% RSLogix 500 project LVD4000_ND_CHICAGO_0020711_Mini.RSS, saved by version 11.00.00.00 %
PROJECT "LVD4000"    % processor: MicroLogix 1400 %

PROGRAM FILES
  LAD 2 "MAIN"  31 rungs  % Main Program Routine %
  LAD 3 "BOT HSC"  2 rungs  % Bottom Conveyor High-Speed Counter Routine %
  LAD 4 "TOP HSC"  2 rungs  % Top Conveyor High-Speed Counter Routine %
  LAD 5 "BOT_TRACK"  3 rungs  % Bottom Conveyor Triggering & Tracking Sequence %
  LAD 6 "TOP_TRACK"  3 rungs  % Top Conveyor Triggering & Tracking Sequence %
  LAD 7 "FOR_HMI"  8 rungs
  LAD 8 "BOT_OPTIC"  6 rungs
  LAD 10 "BOT_TOP"  21 rungs
  LAD 12 "BOT_TRANSF"  3 rungs
  LAD 14 "TOP_OPTIC"  12 rungs
  LAD 16 "TOP_SIDE"  24 rungs
  LAD 18 "TOP_PYRIMI"  5 rungs
  LAD 20 "TOP_TOP"  22 rungs
  LAD 22 "TOP_THREAD"  2 rungs
  LAD 24 "TOP_BLOW"  12 rungs
  LAD 26 "FLOW"  15 rungs
  LAD 28 "FAULTS"  26 rungs
  LAD 30 "SPEED"  8 rungs
  LAD 32 "BOXER"  17 rungs
  LAD 34 "CLEANUP"  20 rungs

DATA FILES
  O0 OUTPUT  6 elements
  I1 INPUT  8 elements
  S2 STATUS  66 elements
  B3 BINARY  11 elements
  T4 TIMER  30 elements
  C5 COUNTER  1 elements
  R6 CONTROL  3 elements
  N7 INTEGER  100 elements
  F8 FLOAT  40 elements
  B9   256 elements
  N10 HMI_COM  100 elements
  B11   256 elements
  B12 BOXER_BITS  3 elements
  N16   1 elements
  B18   11 elements
  T20   1 elements
  R21   4 elements
  B22   35 elements

LADDER 2 "MAIN"    % Main Program Routine %
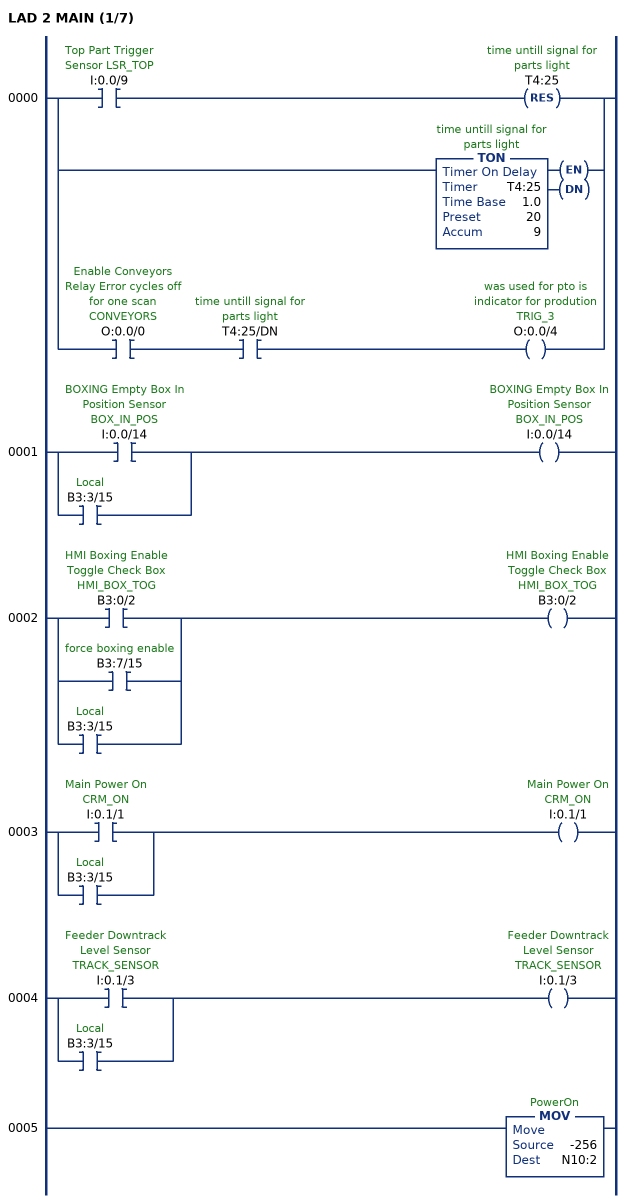
% Rung: 0 %
SOR BST XIC I:0.0/9 RES T4:25 NXB TON T4:25 1.0 20 9 NXB XIC O:0.0/0 XIC T4:25/DN OTE O:0.0/4 BND EOR
%   I:0.0/9  LSR_TOP  "Top Part Trigger Sensor" %
%   T4:25  "time untill signal for parts light" %
%   O:0.0/0  CONVEYORS  "Enable Conveyors Relay Error cycles off for one scan" %
%   O:0.0/4  TRIG_3  "was used for pto is indicator for prodution" %
% Rung: 1 %
SOR BST XIC I:0.0/14 NXB XIC B3:3/15 BND OTE I:0.0/14 EOR
%   I:0.0/14  BOX_IN_POS  "BOXING Empty Box In Position Sensor" %
%   B3:3/15  "Local" %
% Rung: 2 %
SOR BST XIC B3:0/2 NXB XIC B3:7/15 NXB XIC B3:3/15 BND OTE B3:0/2 EOR
%   B3:0/2  HMI_BOX_TOG  "HMI Boxing Enable Toggle Check Box" %
%   B3:7/15  "force boxing enable" %
%   B3:3/15  "Local" %
% Rung: 3 %
SOR BST XIC I:0.1/1 NXB XIC B3:3/15 BND OTE I:0.1/1 EOR
%   I:0.1/1  CRM_ON  "Main Power On" %
%   B3:3/15  "Local" %
% Rung: 4 %
SOR BST XIC I:0.1/3 NXB XIC B3:3/15 BND OTE I:0.1/3 EOR
%   I:0.1/3  TRACK_SENSOR  "Feeder Downtrack Level Sensor" %
%   B3:3/15  "Local" %
% Rung: 5 %
SOR MOV -256 N10:2 EOR
%   N10:2  "PowerOn" %

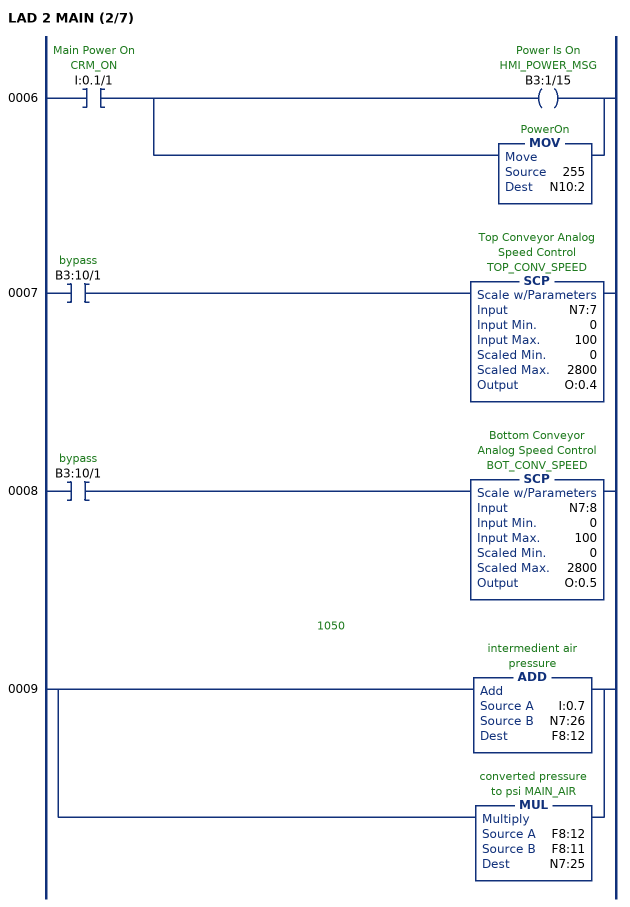
% Rung: 6 %
SOR XIC I:0.1/1 BST OTE B3:1/15 NXB MOV 255 N10:2 BND EOR
%   I:0.1/1  CRM_ON  "Main Power On" %
%   B3:1/15  HMI_POWER_MSG  "Power Is On" %
%   N10:2  "PowerOn" %
% Rung: 7 %
SOR XIC B3:10/1 SCP N7:7 0 100 0 2800 O:0.4 EOR
%   B3:10/1  "bypass" %
%   N7:7  "Top Conv Speed" %
%   O:0.4  TOP_CONV_SPEED  "Top Conveyor Analog Speed Control" %
% Rung: 8 %
SOR XIC B3:10/1 SCP N7:8 0 100 0 2800 O:0.5 EOR
%   B3:10/1  "bypass" %
%   N7:8  "Bottom Conveyor Speed" %
%   O:0.5  BOT_CONV_SPEED  "Bottom Conveyor Analog Speed Control" %
% Rung: 9 %
% 1050 %
SOR BST ADD I:0.7 N7:26 F8:12 NXB MUL F8:12 F8:11 N7:25 BND EOR
%   N7:26  MAIN_AIR_OFFSET  "Main Air Offset" %
%   F8:12  "intermedient air pressure" %
%   F8:11  AIR_MULTIPLIER  "main air multiplyer" %
%   N7:25  MAIN_AIR  "converted pressure to psi" %

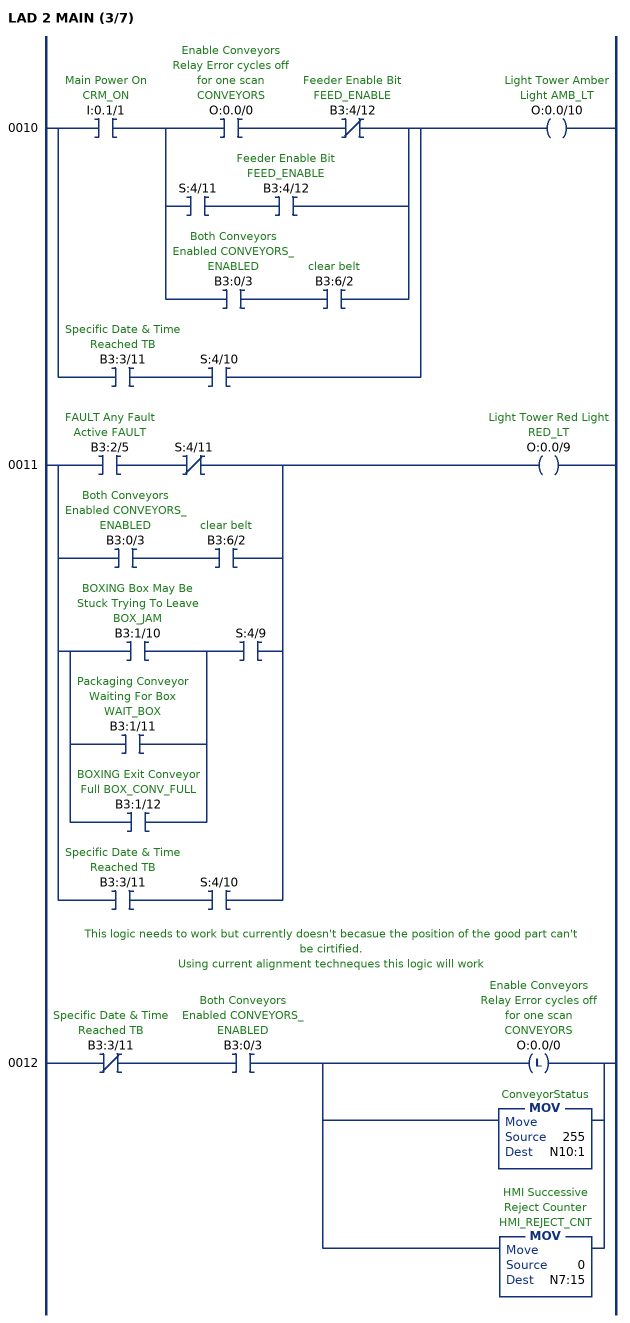
% Rung: 10 %
SOR BST XIC I:0.1/1 BST XIC O:0.0/0 XIO B3:4/12 NXB XIC S:4/11 XIC B3:4/12 NXB XIC B3:0/3 XIC B3:6/2 BND NXB XIC B3:3/11 XIC S:4/10 BND OTE O:0.0/10 EOR
%   I:0.1/1  CRM_ON  "Main Power On" %
%   O:0.0/0  CONVEYORS  "Enable Conveyors Relay Error cycles off for one scan" %
%   B3:4/12  FEED_ENABLE  "Feeder Enable Bit" %
%   B3:0/3  CONVEYORS_ENABLED  "Both Conveyors Enabled" %
%   B3:6/2  "clear belt" %
%   B3:3/11  TB  "Specific Date & Time Reached" %
%   O:0.0/10  AMB_LT  "Light Tower Amber Light" %
% Rung: 11 %
SOR BST BST XIC B3:2/5 XIO S:4/11 NXB XIC B3:0/3 XIC B3:6/2 NXB BST XIC B3:1/10 NXB XIC B3:1/11 NXB XIC B3:1/12 BND XIC S:4/9 BND NXB XIC B3:3/11 XIC S:4/10 BND OTE O:0.0/9 EOR
%   B3:2/5  FAULT  "FAULT Any Fault Active" %
%   B3:0/3  CONVEYORS_ENABLED  "Both Conveyors Enabled" %
%   B3:6/2  "clear belt" %
%   B3:1/10  BOX_JAM  "BOXING Box May Be Stuck Trying To Leave" %
%   B3:1/11  WAIT_BOX  "Packaging Conveyor Waiting For Box" %
%   B3:1/12  BOX_CONV_FULL  "BOXING Exit Conveyor Full" %
%   B3:3/11  TB  "Specific Date & Time Reached" %
%   O:0.0/9  RED_LT  "Light Tower Red Light" %
% Rung: 12 %
% This logic needs to work but currently doesn't becasue the position of the good part can't be cirtified.
% 
% Using current alignment techneques this logic will work %
SOR XIO B3:3/11 XIC B3:0/3 BST OTL O:0.0/0 NXB MOV 255 N10:1 NXB MOV 0 N7:15 BND EOR
%   B3:3/11  TB  "Specific Date & Time Reached" %
%   B3:0/3  CONVEYORS_ENABLED  "Both Conveyors Enabled" %
%   O:0.0/0  CONVEYORS  "Enable Conveyors Relay Error cycles off for one scan" %
%   N10:1  "ConveyorStatus" %
%   N7:15  HMI_REJECT_CNT  "HMI Successive Reject Counter" %

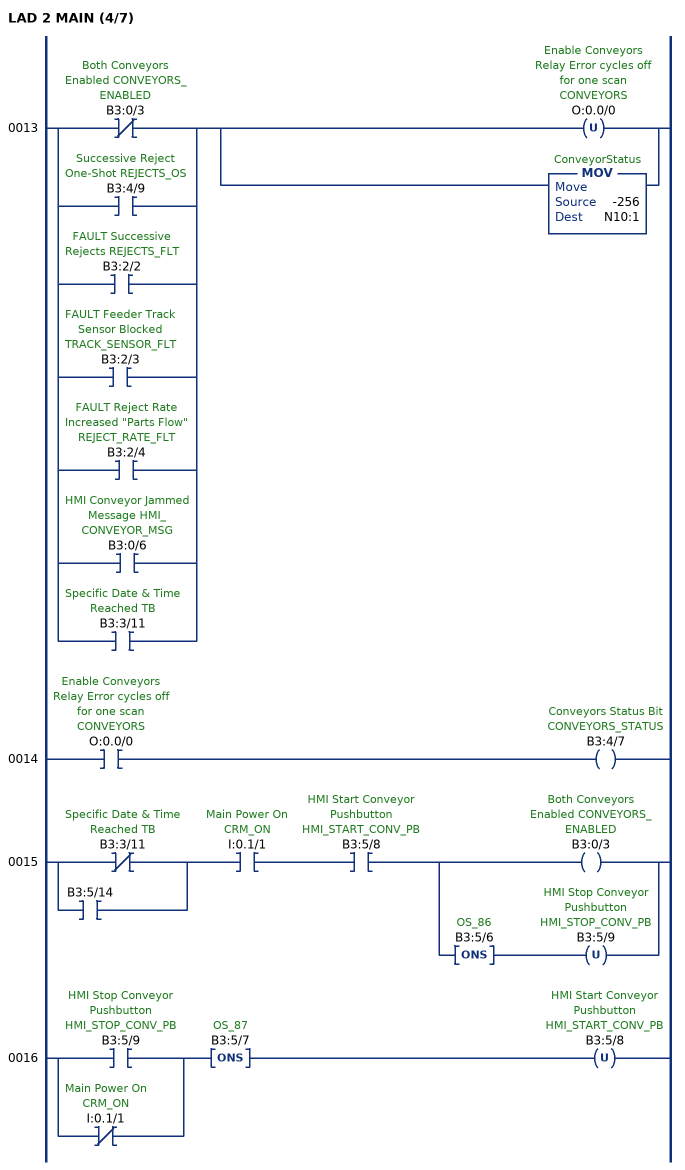
% Rung: 13 %
SOR BST XIO B3:0/3 NXB XIC B3:4/9 NXB XIC B3:2/2 NXB XIC B3:2/3 NXB XIC B3:2/4 NXB XIC B3:0/6 NXB XIC B3:3/11 BND BST OTU O:0.0/0 NXB MOV -256 N10:1 BND EOR
%   B3:0/3  CONVEYORS_ENABLED  "Both Conveyors Enabled" %
%   B3:4/9  REJECTS_OS  "Successive Reject One-Shot" %
%   B3:2/2  REJECTS_FLT  "FAULT Successive Rejects" %
%   B3:2/3  TRACK_SENSOR_FLT  "FAULT Feeder Track Sensor Blocked" %
%   B3:2/4  REJECT_RATE_FLT  "FAULT Reject Rate Increased "Parts Flow"" %
%   B3:0/6  HMI_CONVEYOR_MSG  "HMI Conveyor Jammed Message" %
%   B3:3/11  TB  "Specific Date & Time Reached" %
%   O:0.0/0  CONVEYORS  "Enable Conveyors Relay Error cycles off for one scan" %
%   N10:1  "ConveyorStatus" %
% Rung: 14 %
SOR XIC O:0.0/0 OTE B3:4/7 EOR
%   O:0.0/0  CONVEYORS  "Enable Conveyors Relay Error cycles off for one scan" %
%   B3:4/7  CONVEYORS_STATUS  "Conveyors Status Bit" %
% Rung: 15 %
SOR BST XIO B3:3/11 NXB XIC B3:5/14 BND XIC I:0.1/1 XIC B3:5/8 BST OTE B3:0/3 NXB ONS B3:5/6 OTU B3:5/9 BND EOR
%   B3:3/11  TB  "Specific Date & Time Reached" %
%   I:0.1/1  CRM_ON  "Main Power On" %
%   B3:5/8  HMI_START_CONV_PB  "HMI Start Conveyor Pushbutton" %
%   B3:0/3  CONVEYORS_ENABLED  "Both Conveyors Enabled" %
%   B3:5/6  OS_86 %
%   B3:5/9  HMI_STOP_CONV_PB  "HMI Stop Conveyor Pushbutton" %
% Rung: 16 %
SOR BST XIC B3:5/9 NXB XIO I:0.1/1 BND ONS B3:5/7 OTU B3:5/8 EOR
%   B3:5/9  HMI_STOP_CONV_PB  "HMI Stop Conveyor Pushbutton" %
%   I:0.1/1  CRM_ON  "Main Power On" %
%   B3:5/7  OS_87 %
%   B3:5/8  HMI_START_CONV_PB  "HMI Start Conveyor Pushbutton" %

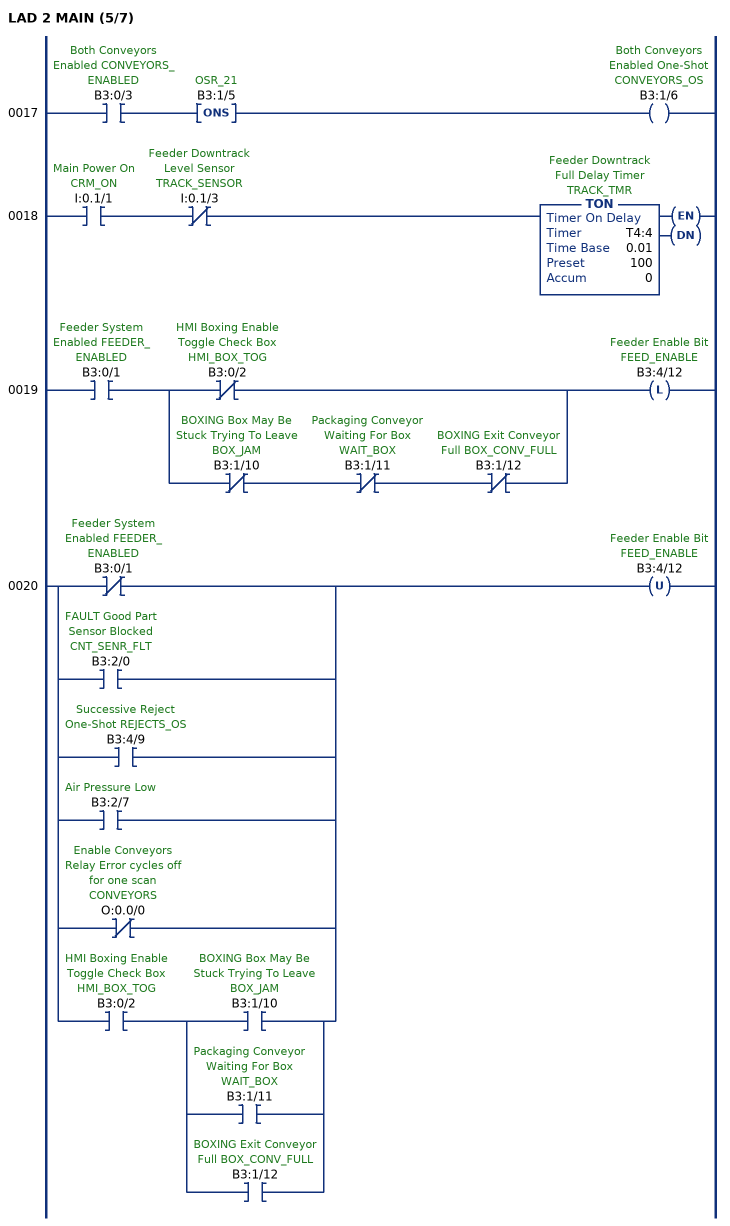
% Rung: 17 %
SOR XIC B3:0/3 ONS B3:1/5 OTE B3:1/6 EOR
%   B3:0/3  CONVEYORS_ENABLED  "Both Conveyors Enabled" %
%   B3:1/5  OSR_21 %
%   B3:1/6  CONVEYORS_OS  "Both Conveyors Enabled One-Shot" %
% Rung: 18 %
SOR XIC I:0.1/1 XIO I:0.1/3 TON T4:4 0.01 100 0 EOR
%   I:0.1/1  CRM_ON  "Main Power On" %
%   I:0.1/3  TRACK_SENSOR  "Feeder Downtrack Level Sensor" %
%   T4:4  TRACK_TMR  "Feeder Downtrack Full Delay Timer" %
% Rung: 19 %
SOR XIC B3:0/1 BST XIO B3:0/2 NXB XIO B3:1/10 XIO B3:1/11 XIO B3:1/12 BND OTL B3:4/12 EOR
%   B3:0/1  FEEDER_ENABLED  "Feeder System Enabled" %
%   B3:0/2  HMI_BOX_TOG  "HMI Boxing Enable Toggle Check Box" %
%   B3:1/10  BOX_JAM  "BOXING Box May Be Stuck Trying To Leave" %
%   B3:1/11  WAIT_BOX  "Packaging Conveyor Waiting For Box" %
%   B3:1/12  BOX_CONV_FULL  "BOXING Exit Conveyor Full" %
%   B3:4/12  FEED_ENABLE  "Feeder Enable Bit" %
% Rung: 20 %
SOR BST XIO B3:0/1 NXB XIC B3:2/0 NXB XIC B3:4/9 NXB XIC B3:2/7 NXB XIO O:0.0/0 NXB XIC B3:0/2 BST XIC B3:1/10 NXB XIC B3:1/11 NXB XIC B3:1/12 BND BND OTU B3:4/12 EOR
%   B3:0/1  FEEDER_ENABLED  "Feeder System Enabled" %
%   B3:2/0  CNT_SENR_FLT  "FAULT Good Part Sensor Blocked" %
%   B3:4/9  REJECTS_OS  "Successive Reject One-Shot" %
%   B3:2/7  "Air Pressure Low" %
%   O:0.0/0  CONVEYORS  "Enable Conveyors Relay Error cycles off for one scan" %
%   B3:0/2  HMI_BOX_TOG  "HMI Boxing Enable Toggle Check Box" %
%   B3:1/10  BOX_JAM  "BOXING Box May Be Stuck Trying To Leave" %
%   B3:1/11  WAIT_BOX  "Packaging Conveyor Waiting For Box" %
%   B3:1/12  BOX_CONV_FULL  "BOXING Exit Conveyor Full" %
%   B3:4/12  FEED_ENABLE  "Feeder Enable Bit" %

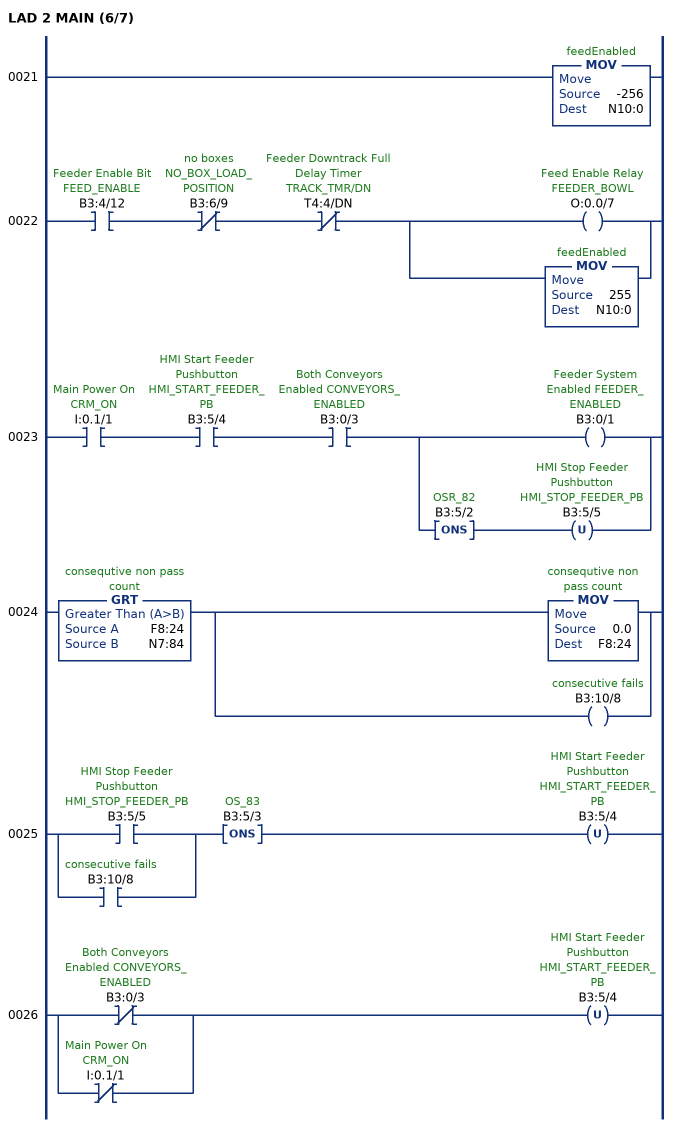
% Rung: 21 %
SOR MOV -256 N10:0 EOR
%   N10:0  "feedEnabled" %
% Rung: 22 %
SOR XIC B3:4/12 XIO B3:6/9 XIO T4:4/DN BST OTE O:0.0/7 NXB MOV 255 N10:0 BND EOR
%   B3:4/12  FEED_ENABLE  "Feeder Enable Bit" %
%   B3:6/9  NO_BOX_LOAD_POSITION  "no boxes" %
%   T4:4  TRACK_TMR  "Feeder Downtrack Full Delay Timer" %
%   O:0.0/7  FEEDER_BOWL  "Feed Enable Relay" %
%   N10:0  "feedEnabled" %
% Rung: 23 %
SOR XIC I:0.1/1 XIC B3:5/4 XIC B3:0/3 BST OTE B3:0/1 NXB ONS B3:5/2 OTU B3:5/5 BND EOR
%   I:0.1/1  CRM_ON  "Main Power On" %
%   B3:5/4  HMI_START_FEEDER_PB  "HMI Start Feeder Pushbutton" %
%   B3:0/3  CONVEYORS_ENABLED  "Both Conveyors Enabled" %
%   B3:0/1  FEEDER_ENABLED  "Feeder System Enabled" %
%   B3:5/2  OSR_82 %
%   B3:5/5  HMI_STOP_FEEDER_PB  "HMI Stop Feeder Pushbutton" %
% Rung: 24 %
SOR GRT F8:24 N7:84 BST MOV 0.0 F8:24 NXB OTE B3:10/8 BND EOR
%   F8:24  "consequtive non pass count" %
%   B3:10/8  "consecutive fails" %
% Rung: 25 %
SOR BST XIC B3:5/5 NXB XIC B3:10/8 BND ONS B3:5/3 OTU B3:5/4 EOR
%   B3:5/5  HMI_STOP_FEEDER_PB  "HMI Stop Feeder Pushbutton" %
%   B3:10/8  "consecutive fails" %
%   B3:5/3  OS_83 %
%   B3:5/4  HMI_START_FEEDER_PB  "HMI Start Feeder Pushbutton" %
% Rung: 26 %
SOR BST XIO B3:0/3 NXB XIO I:0.1/1 BND OTU B3:5/4 EOR
%   B3:0/3  CONVEYORS_ENABLED  "Both Conveyors Enabled" %
%   I:0.1/1  CRM_ON  "Main Power On" %
%   B3:5/4  HMI_START_FEEDER_PB  "HMI Start Feeder Pushbutton" %

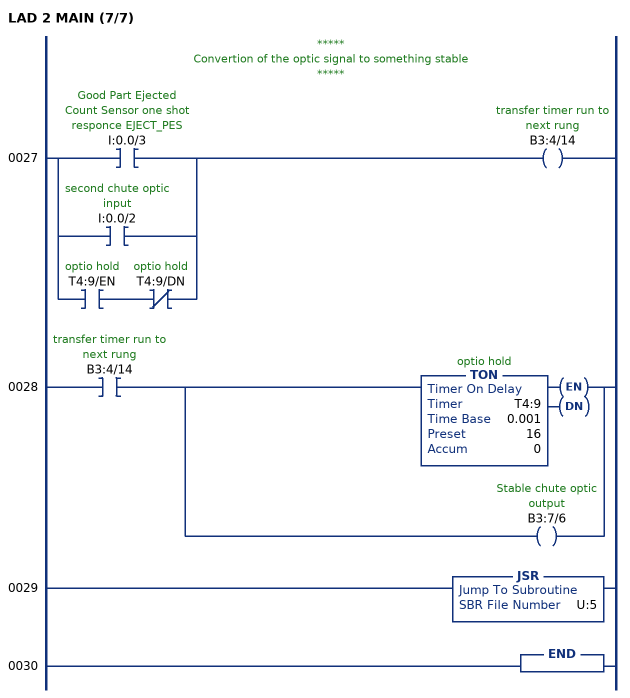
% Rung: 27 %
% *****
% 
% Convertion of the optic signal to something stable
% 
% ***** %
SOR BST XIC I:0.0/3 NXB XIC I:0.0/2 NXB XIC T4:9/EN XIO T4:9/DN BND OTE B3:4/14 EOR
%   I:0.0/3  EJECT_PES  "Good Part Ejected Count Sensor one shot responce" %
%   I:0.0/2  "second chute optic input" %
%   T4:9  "optio hold" %
%   B3:4/14  "transfer timer run to next rung" %
% Rung: 28 %
SOR XIC B3:4/14 BST TON T4:9 0.001 16 0 NXB OTE B3:7/6 BND EOR
%   B3:4/14  "transfer timer run to next rung" %
%   T4:9  "optio hold" %
%   B3:7/6  "Stable chute optic output" %
% Rung: 29 %
SOR JSR U:5 EOR
% Rung: 30 %
SOR END EOR

LADDER 3 "BOT HSC"    % Bottom Conveyor High-Speed Counter Routine %
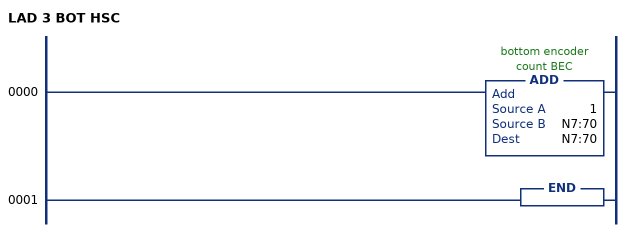
% Rung: 0 %
SOR ADD 1 N7:70 N7:70 EOR
%   N7:70  BEC  "bottom encoder count" %
% Rung: 1 %
SOR END EOR

LADDER 4 "TOP HSC"    % Top Conveyor High-Speed Counter Routine %
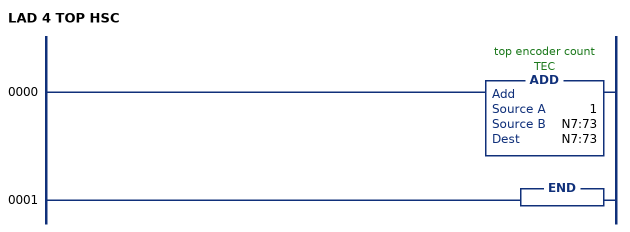
% Rung: 0 %
SOR ADD 1 N7:73 N7:73 EOR
%   N7:73  TEC  "top encoder count" %
% Rung: 1 %
SOR END EOR

LADDER 5 "BOT_TRACK"    % Bottom Conveyor Triggering & Tracking Sequence %
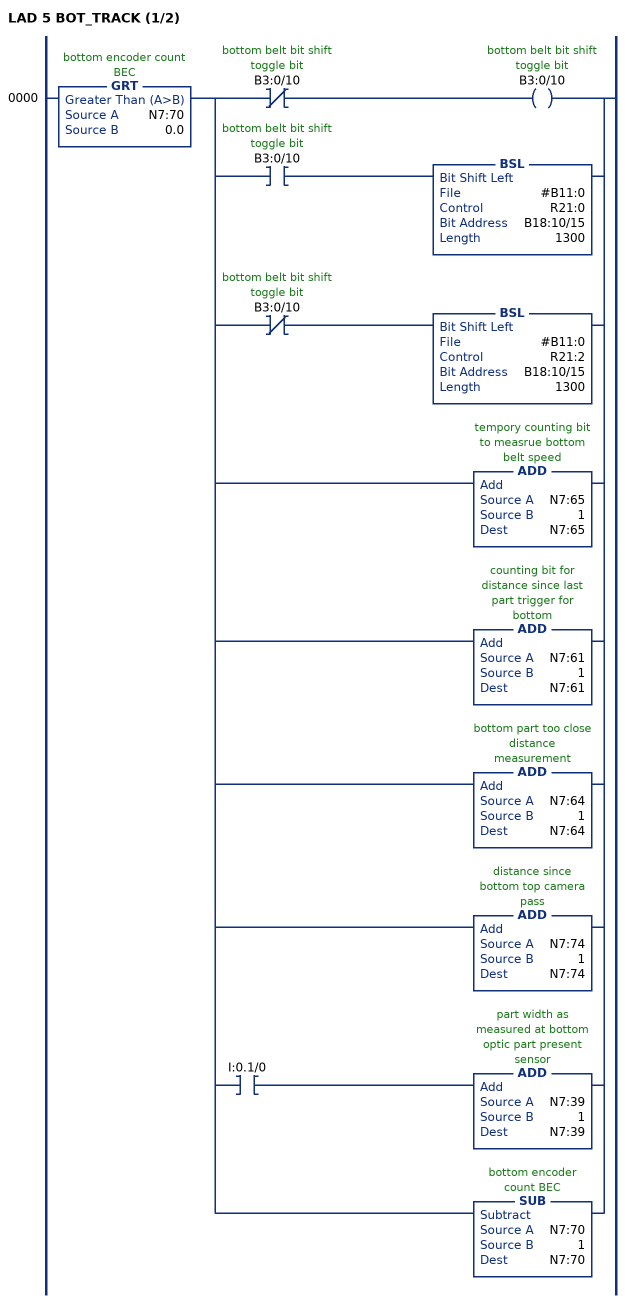
% Rung: 0 %
SOR GRT N7:70 0.0 BST XIO B3:0/10 OTE B3:0/10 NXB XIC B3:0/10 BSL #B11:0 R21:0 B18:10/15 1300 NXB XIO B3:0/10 BSL #B11:0 R21:2 B18:10/15 1300 NXB ADD N7:65 1 N7:65 NXB ADD N7:61 1 N7:61 NXB ADD N7:64 1 N7:64 NXB ADD N7:74 1 N7:74 NXB XIC I:0.1/0 ADD N7:39 1 N7:39 NXB SUB N7:70 1 N7:70 BND EOR
%   N7:70  BEC  "bottom encoder count" %
%   B3:0/10  "bottom belt bit shift toggle bit" %
%   R21:0  "Trigger Shift Register" %
%   B18:10/15  "Reserved For Shift Registers" %
%   N7:65  "tempory counting bit to measrue bottom belt speed" %
%   N7:61  "counting bit for distance since last part trigger for bottom" %
%   N7:64  "bottom part too close distance measurement" %
%   N7:74  "distance since bottom top camera pass" %
%   N7:39  "part width as measured at bottom optic part present sensor" %

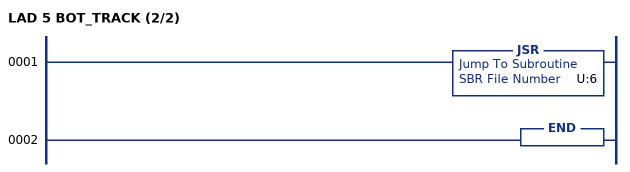
% Rung: 1 %
SOR JSR U:6 EOR
% Rung: 2 %
SOR END EOR

LADDER 6 "TOP_TRACK"    % Top Conveyor Triggering & Tracking Sequence %
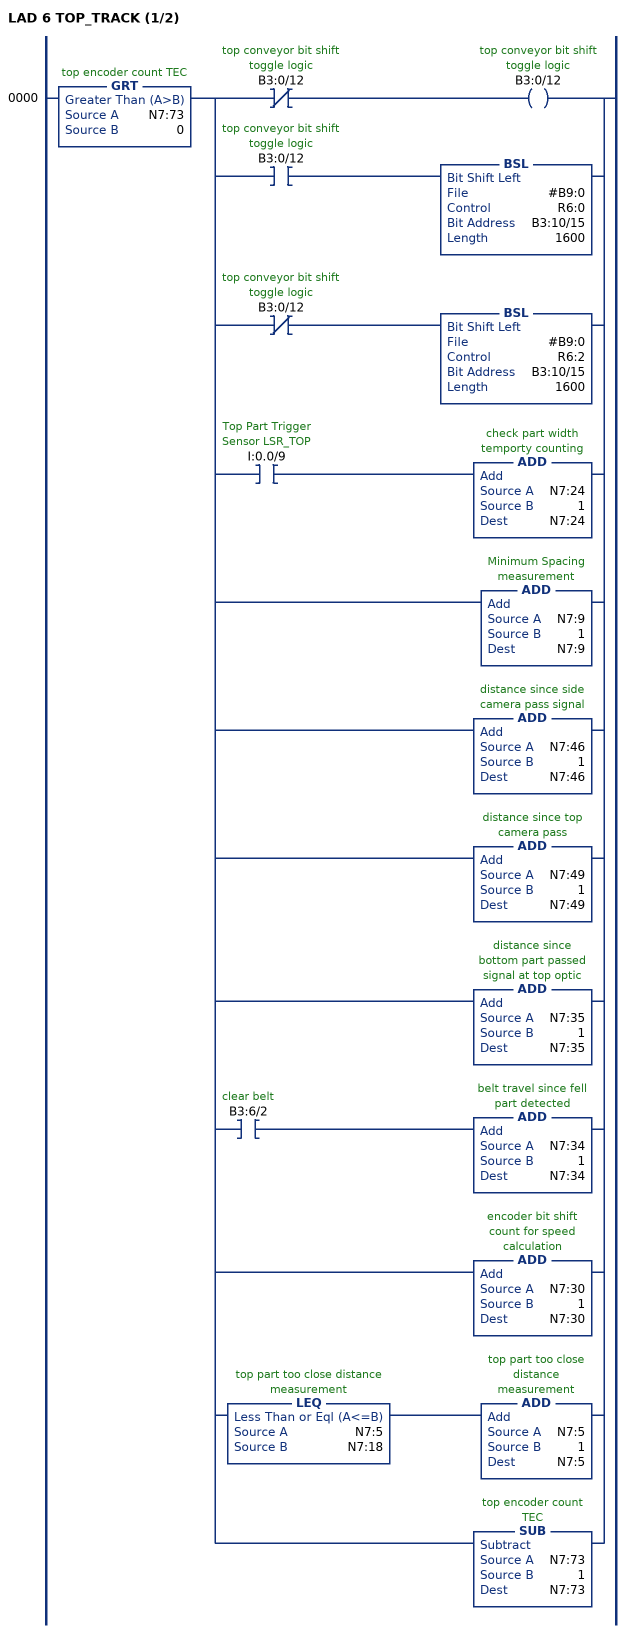
% Rung: 0 %
SOR GRT N7:73 0 BST XIO B3:0/12 OTE B3:0/12 NXB XIC B3:0/12 BSL #B9:0 R6:0 B3:10/15 1600 NXB XIO B3:0/12 BSL #B9:0 R6:2 B3:10/15 1600 NXB XIC I:0.0/9 ADD N7:24 1 N7:24 NXB ADD N7:9 1 N7:9 NXB ADD N7:46 1 N7:46 NXB ADD N7:49 1 N7:49 NXB ADD N7:35 1 N7:35 NXB XIC B3:6/2 ADD N7:34 1 N7:34 NXB ADD N7:30 1 N7:30 NXB LEQ N7:5 N7:18 ADD N7:5 1 N7:5 NXB SUB N7:73 1 N7:73 BND EOR
%   N7:73  TEC  "top encoder count" %
%   B3:0/12  "top conveyor bit shift toggle logic" %
%   R6:0  "Top Conveyor Part Tracking Bit Shit" %
%   B3:10/15  "Reserved For Shift Registers" %
%   I:0.0/9  LSR_TOP  "Top Part Trigger Sensor" %
%   N7:24  "check part width temporty counting" %
%   N7:9  "Minimum Spacing measurement" %
%   N7:46  "distance since side camera pass signal" %
%   N7:49  "distance since top camera pass" %
%   N7:35  "distance since bottom part passed signal at top optic" %
%   B3:6/2  "clear belt" %
%   N7:34  "belt travel since fell part detected" %
%   N7:30  "encoder bit shift count for speed calculation" %
%   N7:5  "top part too close distance measurement" %
%   N7:18  "total distance to remove part present signals when parts are too close top" %

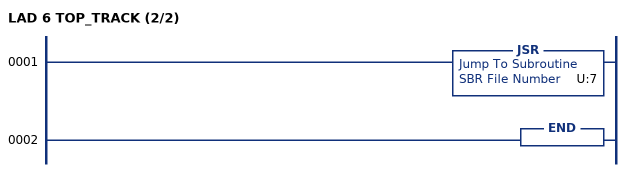
% Rung: 1 %
SOR JSR U:7 EOR
% Rung: 2 %
SOR END EOR

LADDER 7 "FOR_HMI"
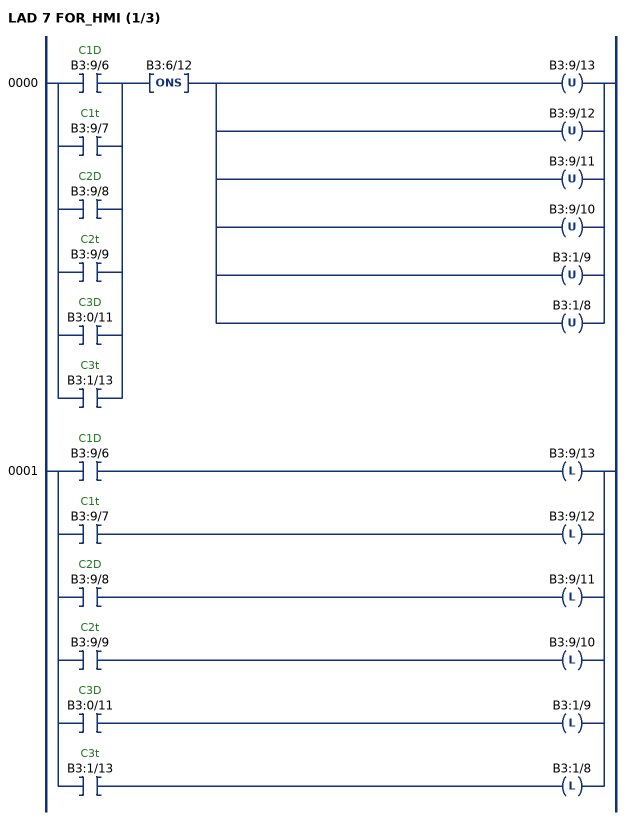
% Rung: 0 %
SOR BST XIC B3:9/6 NXB XIC B3:9/7 NXB XIC B3:9/8 NXB XIC B3:9/9 NXB XIC B3:0/11 NXB XIC B3:1/13 BND ONS B3:6/12 BST OTU B3:9/13 NXB OTU B3:9/12 NXB OTU B3:9/11 NXB OTU B3:9/10 NXB OTU B3:1/9 NXB OTU B3:1/8 BND EOR
%   B3:9/6  "C1D" %
%   B3:9/7  "C1t" %
%   B3:9/8  "C2D" %
%   B3:9/9  "C2t" %
%   B3:0/11  "C3D" %
%   B3:1/13  "C3t" %
% Rung: 1 %
SOR BST XIC B3:9/6 OTL B3:9/13 NXB XIC B3:9/7 OTL B3:9/12 NXB XIC B3:9/8 OTL B3:9/11 NXB XIC B3:9/9 OTL B3:9/10 NXB XIC B3:0/11 OTL B3:1/9 NXB XIC B3:1/13 OTL B3:1/8 BND EOR
%   B3:9/6  "C1D" %
%   B3:9/7  "C1t" %
%   B3:9/8  "C2D" %
%   B3:9/9  "C2t" %
%   B3:0/11  "C3D" %
%   B3:1/13  "C3t" %

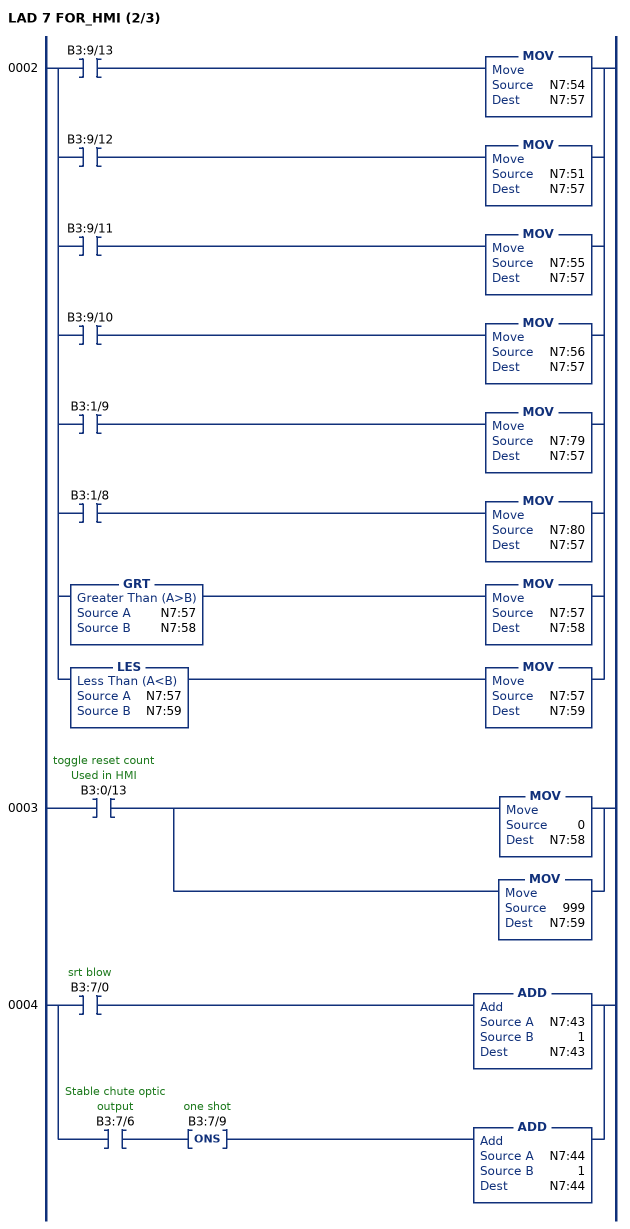
% Rung: 2 %
SOR BST XIC B3:9/13 MOV N7:54 N7:57 NXB XIC B3:9/12 MOV N7:51 N7:57 NXB XIC B3:9/11 MOV N7:55 N7:57 NXB XIC B3:9/10 MOV N7:56 N7:57 NXB XIC B3:1/9 MOV N7:79 N7:57 NXB XIC B3:1/8 MOV N7:80 N7:57 NXB GRT N7:57 N7:58 MOV N7:57 N7:58 NXB LES N7:57 N7:59 MOV N7:57 N7:59 BND EOR
%   N7:54  "side camera responce distance" %
%   N7:51  "side camera response time ms" %
%   N7:55  "top camera responce distance" %
%   N7:56  "top camera responce time ms" %
%   N7:79  "bottom top camera responce distance" %
%   N7:80  "bottom top camera responce time" %
% Rung: 3 %
SOR XIC B3:0/13 BST MOV 0 N7:58 NXB MOV 999 N7:59 BND EOR
%   B3:0/13  "toggle reset count Used in HMI" %
% Rung: 4 %
SOR BST XIC B3:7/0 ADD N7:43 1 N7:43 NXB XIC B3:7/6 ONS B3:7/9 ADD N7:44 1 N7:44 BND EOR
%   B3:7/0  "srt blow" %
%   B3:7/6  "Stable chute optic output" %
%   B3:7/9  "one shot" %

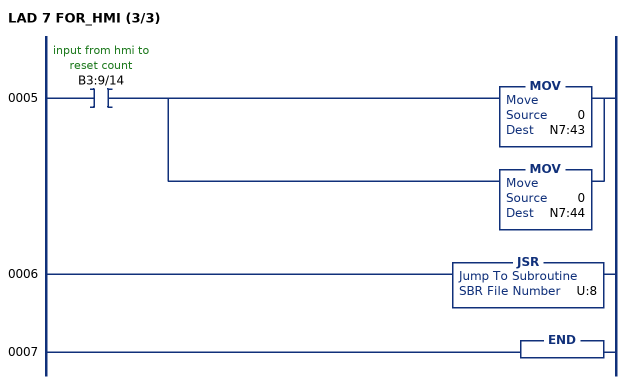
% Rung: 5 %
SOR XIC B3:9/14 BST MOV 0 N7:43 NXB MOV 0 N7:44 BND EOR
%   B3:9/14  "input from hmi to reset count" %
% Rung: 6 %
SOR JSR U:8 EOR
% Rung: 7 %
SOR END EOR

LADDER 8 "BOT_OPTIC"
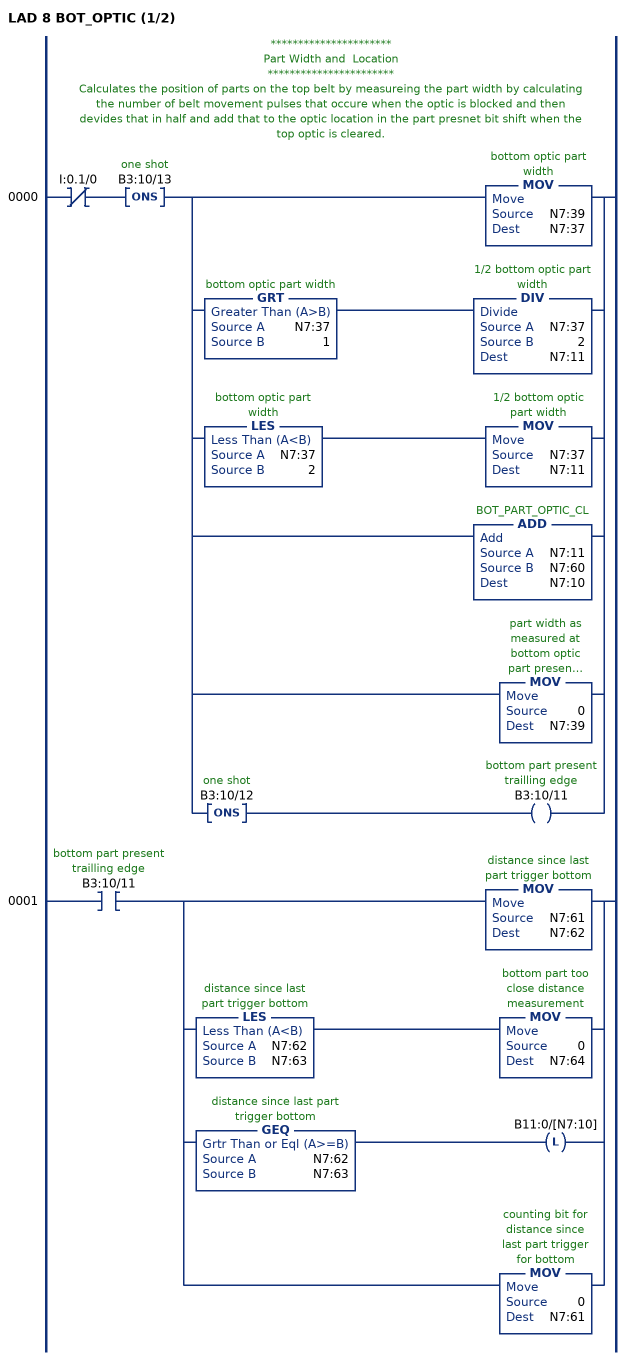
% Rung: 0 %
%  **********************
% Part Width and  Location
% ***********************
% 
% Calculates the position of parts on the top belt by measureing the part width by calculating the number of belt movement pulses that occure when the optic is blocked and then devides that in half and add that to the optic location in the part presnet bit shift when the top optic is cleared. %
SOR XIO I:0.1/0 ONS B3:10/13 BST MOV N7:39 N7:37 NXB GRT N7:37 1 DIV N7:37 2 N7:11 NXB LES N7:37 2 MOV N7:37 N7:11 NXB ADD N7:11 N7:60 N7:10 NXB MOV 0 N7:39 NXB ONS B3:10/12 OTE B3:10/11 BND EOR
%   B3:10/13  "one shot" %
%   N7:39  "part width as measured at bottom optic part present sensor" %
%   N7:37  "bottom optic part width" %
%   N7:11  "1/2 bottom optic part width" %
%   N7:60  "bottom optic location" %
%   N7:10  BOT_PART_OPTIC_CL %
%   B3:10/12  "one shot" %
%   B3:10/11  "bottom part present trailling edge" %
% Rung: 1 %
SOR XIC B3:10/11 BST MOV N7:61 N7:62 NXB LES N7:62 N7:63 MOV 0 N7:64 NXB GEQ N7:62 N7:63 OTL B11:0/[N7:10] NXB MOV 0 N7:61 BND EOR
%   B3:10/11  "bottom part present trailling edge" %
%   N7:61  "counting bit for distance since last part trigger for bottom" %
%   N7:62  "distance since last part trigger bottom" %
%   N7:63  "min part spacing bottom" %
%   N7:64  "bottom part too close distance measurement" %
%   N7:10  BOT_PART_OPTIC_CL %

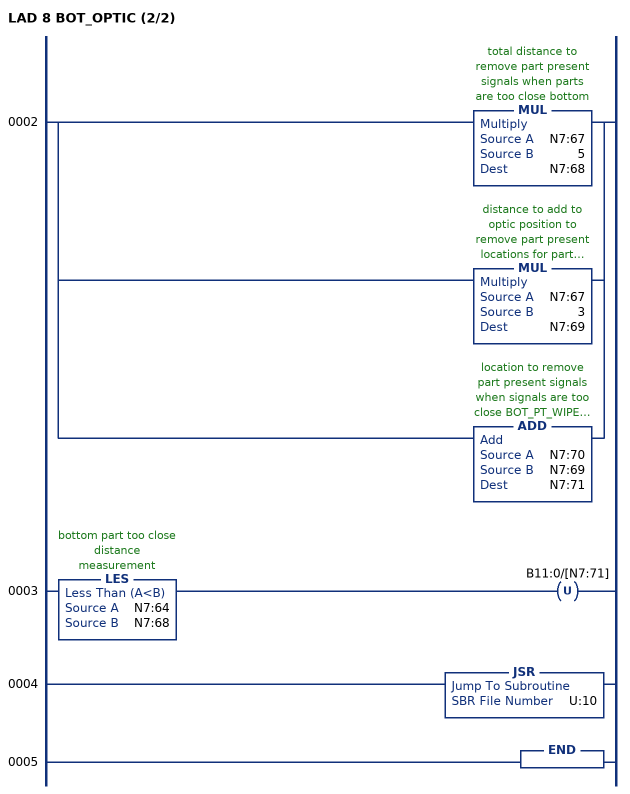
% Rung: 2 %
SOR BST MUL N7:67 5 N7:68 NXB MUL N7:67 3 N7:69 NXB ADD N7:70 N7:69 N7:71 BND EOR
%   N7:67  "distance to remove trigger signals when part spacing too close bottom" %
%   N7:68  "total distance to remove part present signals when parts are too close bottom" %
%   N7:69  "distance to add to optic position to remove part present locations for parts too close bottom" %
%   N7:70  BEC  "bottom encoder count" %
%   N7:71  BOT_PT_WIPE_LOC  "location to remove part present signals when signals are too close" %
% Rung: 3 %
SOR LES N7:64 N7:68 OTU B11:0/[N7:71] EOR
%   N7:64  "bottom part too close distance measurement" %
%   N7:68  "total distance to remove part present signals when parts are too close bottom" %
%   N7:71  BOT_PT_WIPE_LOC  "location to remove part present signals when signals are too close" %
% Rung: 4 %
SOR JSR U:10 EOR
% Rung: 5 %
SOR END EOR

LADDER 10 "BOT_TOP"
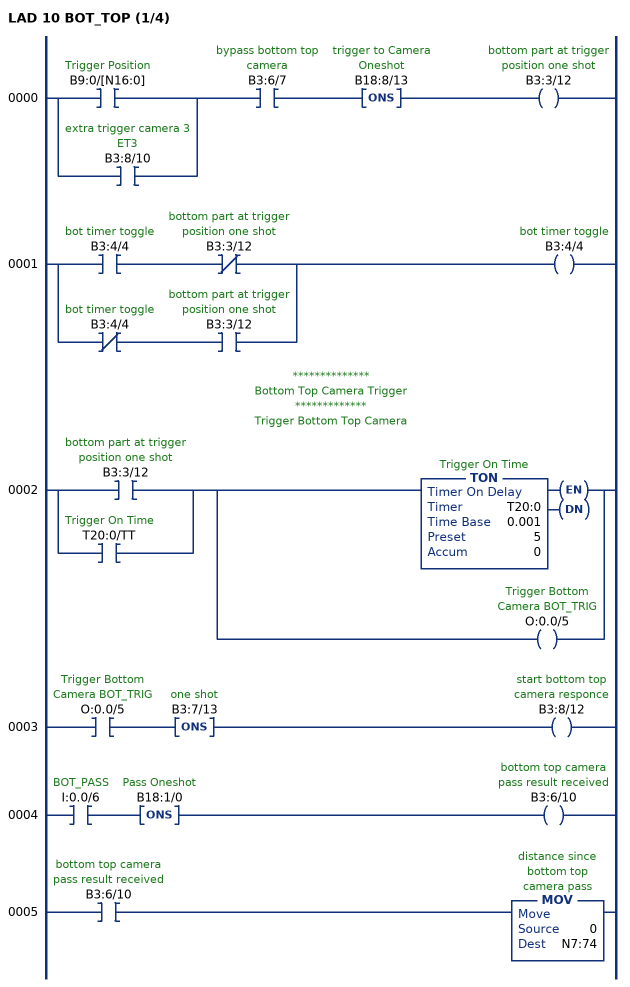
% Rung: 0 %
SOR BST XIC B9:0/[N16:0] NXB XIC B3:8/10 BND XIC B3:6/7 ONS B18:8/13 OTE B3:3/12 EOR
%   B9:0/[N16:0]  "Trigger Position" %
%   N16:0  BOT_TRIGGER  "Trigger Position" %
%   B3:8/10  ET3  "extra trigger camera 3" %
%   B3:6/7  "bypass bottom top camera" %
%   B18:8/13  "trigger to Camera Oneshot" %
%   B3:3/12  "bottom part at trigger position one shot" %
% Rung: 1 %
SOR BST XIC B3:4/4 XIO B3:3/12 NXB XIO B3:4/4 XIC B3:3/12 BND OTE B3:4/4 EOR
%   B3:4/4  "bot timer toggle" %
%   B3:3/12  "bottom part at trigger position one shot" %
% Rung: 2 %
% **************
% Bottom Top Camera Trigger
% *************
% 
% Trigger Bottom Top Camera %
SOR BST XIC B3:3/12 NXB XIC T20:0/TT BND BST TON T20:0 0.001 5 0 NXB OTE O:0.0/5 BND EOR
%   B3:3/12  "bottom part at trigger position one shot" %
%   T20:0  "Trigger On Time" %
%   O:0.0/5  BOT_TRIG  "Trigger Bottom Camera" %
% Rung: 3 %
SOR XIC O:0.0/5 ONS B3:7/13 OTE B3:8/12 EOR
%   O:0.0/5  BOT_TRIG  "Trigger Bottom Camera" %
%   B3:7/13  "one shot" %
%   B3:8/12  "start bottom top camera responce" %
% Rung: 4 %
SOR XIC I:0.0/6 ONS B18:1/0 OTE B3:6/10 EOR
%   I:0.0/6  BOT_PASS %
%   B18:1/0  "Pass Oneshot" %
%   B3:6/10  "bottom top camera pass result received" %
% Rung: 5 %
SOR XIC B3:6/10 MOV 0 N7:74 EOR
%   B3:6/10  "bottom top camera pass result received" %
%   N7:74  "distance since bottom top camera pass" %

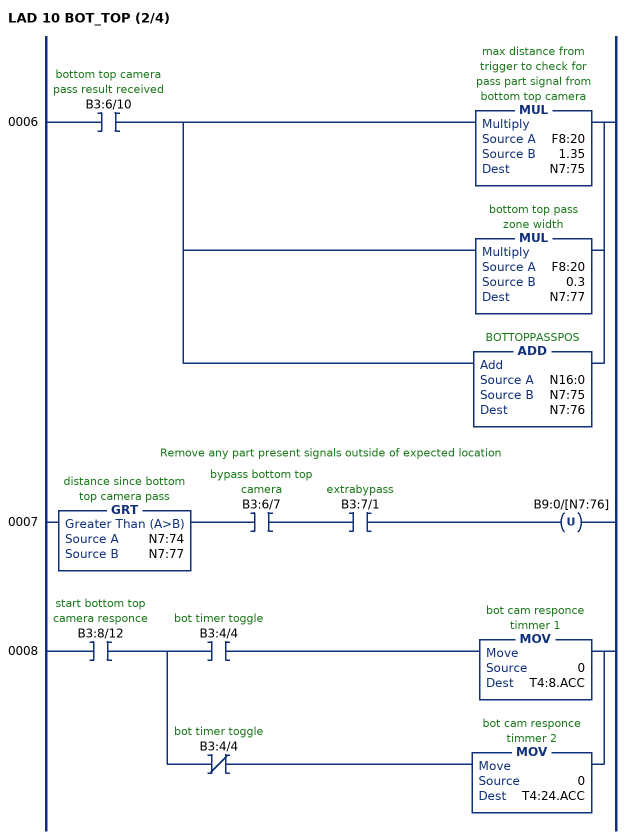
% Rung: 6 %
SOR XIC B3:6/10 BST MUL F8:20 1.35 N7:75 NXB MUL F8:20 0.3 N7:77 NXB ADD N16:0 N7:75 N7:76 BND EOR
%   B3:6/10  "bottom top camera pass result received" %
%   F8:20  "bot belt speed average in pulses per 100ms" %
%   N7:75  "max distance from trigger to check for pass part signal from bottom top camera" %
%   N7:77  "bottom top pass zone width" %
%   N16:0  BOT_TRIGGER  "Trigger Position" %
%   N7:76  BOTTOPPASSPOS %
% Rung: 7 %
% Remove any part present signals outside of expected location %
SOR GRT N7:74 N7:77 XIC B3:6/7 XIC B3:7/1 OTU B9:0/[N7:76] EOR
%   N7:74  "distance since bottom top camera pass" %
%   N7:77  "bottom top pass zone width" %
%   B3:6/7  "bypass bottom top camera" %
%   B3:7/1  "extrabypass" %
%   N7:76  BOTTOPPASSPOS %
% Rung: 8 %
SOR XIC B3:8/12 BST XIC B3:4/4 MOV 0 T4:8.ACC NXB XIO B3:4/4 MOV 0 T4:24.ACC BND EOR
%   B3:8/12  "start bottom top camera responce" %
%   B3:4/4  "bot timer toggle" %
%   T4:8  "bot cam responce timmer 1" %
%   T4:24  "bot cam responce timmer 2" %

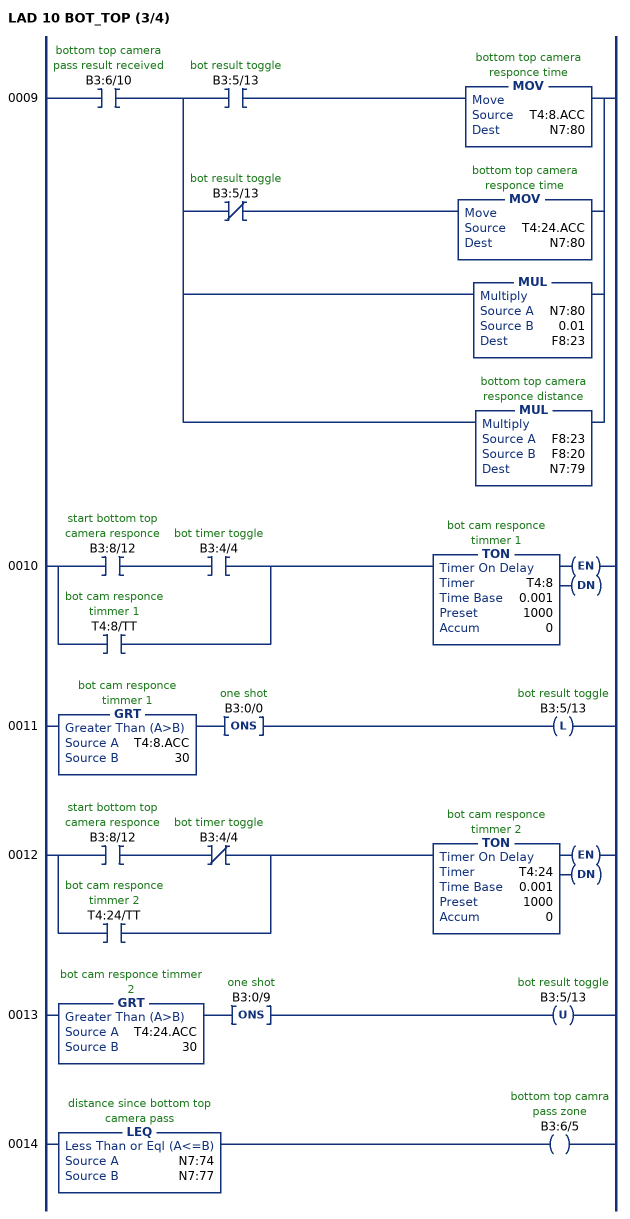
% Rung: 9 %
SOR XIC B3:6/10 BST XIC B3:5/13 MOV T4:8.ACC N7:80 NXB XIO B3:5/13 MOV T4:24.ACC N7:80 NXB MUL N7:80 0.01 F8:23 NXB MUL F8:23 F8:20 N7:79 BND EOR
%   B3:6/10  "bottom top camera pass result received" %
%   B3:5/13  "bot result toggle" %
%   T4:8  "bot cam responce timmer 1" %
%   N7:80  "bottom top camera responce time" %
%   T4:24  "bot cam responce timmer 2" %
%   F8:20  "bot belt speed average in pulses per 100ms" %
%   N7:79  "bottom top camera responce distance" %
% Rung: 10 %
SOR BST XIC B3:8/12 XIC B3:4/4 NXB XIC T4:8/TT BND TON T4:8 0.001 1000 0 EOR
%   B3:8/12  "start bottom top camera responce" %
%   B3:4/4  "bot timer toggle" %
%   T4:8  "bot cam responce timmer 1" %
% Rung: 11 %
SOR GRT T4:8.ACC 30 ONS B3:0/0 OTL B3:5/13 EOR
%   T4:8  "bot cam responce timmer 1" %
%   B3:0/0  "one shot" %
%   B3:5/13  "bot result toggle" %
% Rung: 12 %
SOR BST XIC B3:8/12 XIO B3:4/4 NXB XIC T4:24/TT BND TON T4:24 0.001 1000 0 EOR
%   B3:8/12  "start bottom top camera responce" %
%   B3:4/4  "bot timer toggle" %
%   T4:24  "bot cam responce timmer 2" %
% Rung: 13 %
SOR GRT T4:24.ACC 30 ONS B3:0/9 OTU B3:5/13 EOR
%   T4:24  "bot cam responce timmer 2" %
%   B3:0/9  "one shot" %
%   B3:5/13  "bot result toggle" %
% Rung: 14 %
SOR LEQ N7:74 N7:77 OTE B3:6/5 EOR
%   N7:74  "distance since bottom top camera pass" %
%   N7:77  "bottom top pass zone width" %
%   B3:6/5  "bottom top camra pass zone" %

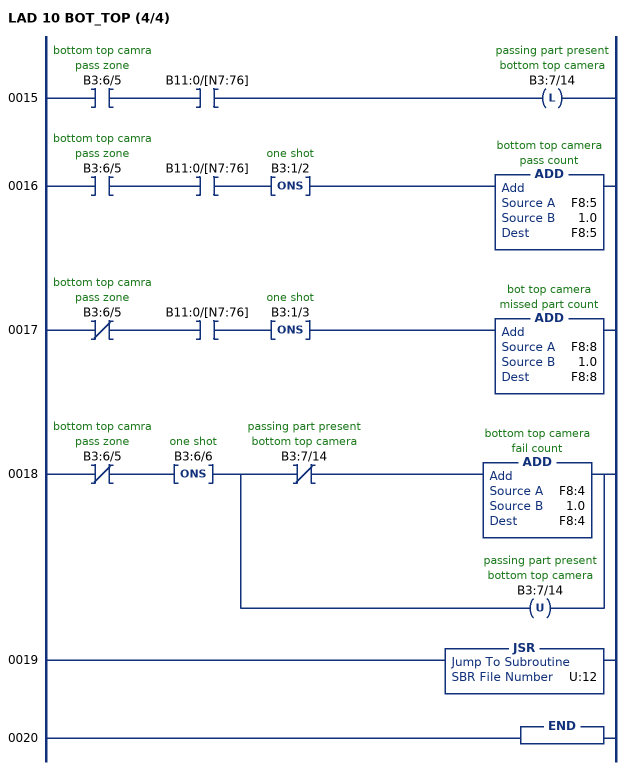
% Rung: 15 %
SOR XIC B3:6/5 XIC B11:0/[N7:76] OTL B3:7/14 EOR
%   B3:6/5  "bottom top camra pass zone" %
%   N7:76  BOTTOPPASSPOS %
%   B3:7/14  "passing part present bottom top camera" %
% Rung: 16 %
SOR XIC B3:6/5 XIC B11:0/[N7:76] ONS B3:1/2 ADD F8:5 1.0 F8:5 EOR
%   B3:6/5  "bottom top camra pass zone" %
%   N7:76  BOTTOPPASSPOS %
%   B3:1/2  "one shot" %
%   F8:5  "bottom top camera pass count" %
% Rung: 17 %
SOR XIO B3:6/5 XIC B11:0/[N7:76] ONS B3:1/3 ADD F8:8 1.0 F8:8 EOR
%   B3:6/5  "bottom top camra pass zone" %
%   N7:76  BOTTOPPASSPOS %
%   B3:1/3  "one shot" %
%   F8:8  "bot top camera missed part count" %
% Rung: 18 %
SOR XIO B3:6/5 ONS B3:6/6 BST XIO B3:7/14 ADD F8:4 1.0 F8:4 NXB OTU B3:7/14 BND EOR
%   B3:6/5  "bottom top camra pass zone" %
%   B3:6/6  "one shot" %
%   B3:7/14  "passing part present bottom top camera" %
%   F8:4  "bottom top camera fail count" %
% Rung: 19 %
SOR JSR U:12 EOR
% Rung: 20 %
SOR END EOR

LADDER 12 "BOT_TRANSF"
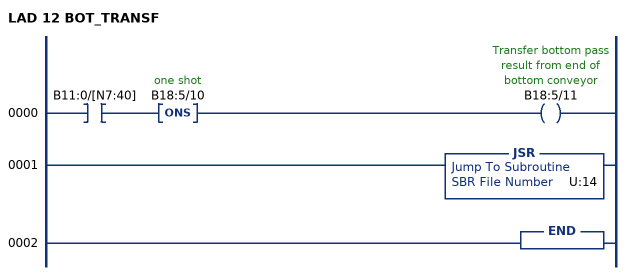
% Rung: 0 %
SOR XIC B11:0/[N7:40] ONS B18:5/10 OTE B18:5/11 EOR
%   N7:40  BOT_TRANS_POS  "bottom conveyor pass signal transfer position" %
%   B18:5/10  "one shot" %
%   B18:5/11  "Transfer bottom pass result from end of bottom conveyor" %
% Rung: 1 %
SOR JSR U:14 EOR
% Rung: 2 %
SOR END EOR

LADDER 14 "TOP_OPTIC"
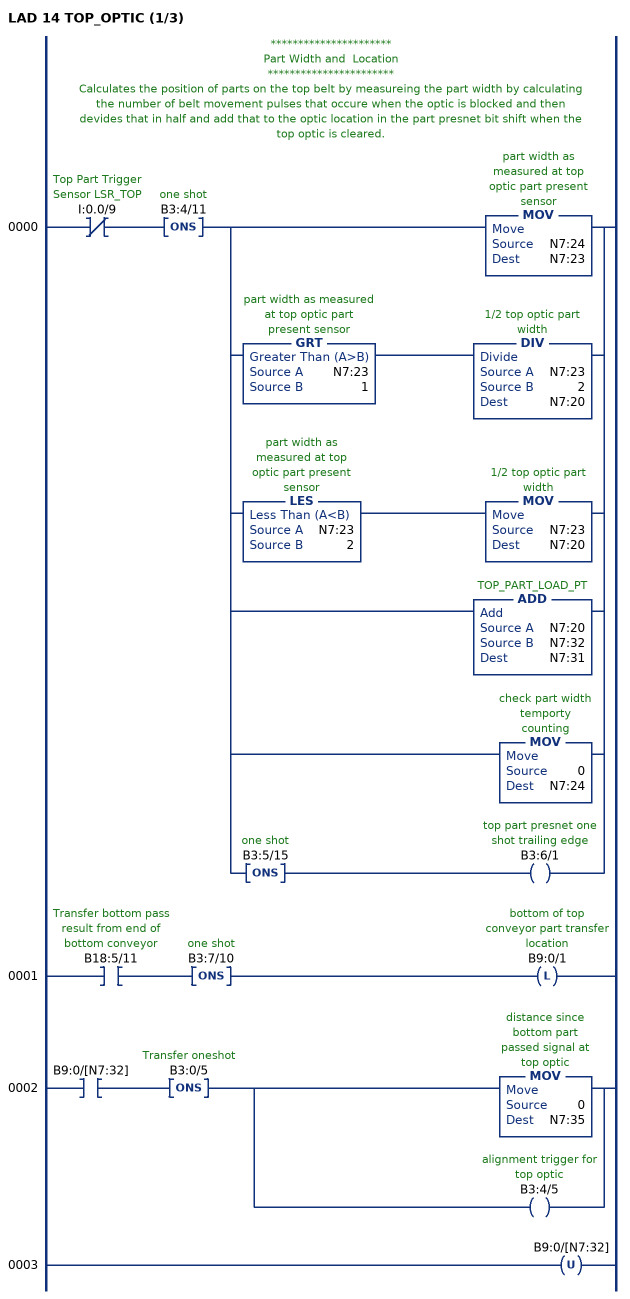
% Rung: 0 %
%  **********************
% Part Width and  Location
% ***********************
% 
% Calculates the position of parts on the top belt by measureing the part width by calculating the number of belt movement pulses that occure when the optic is blocked and then devides that in half and add that to the optic location in the part presnet bit shift when the top optic is cleared. %
SOR XIO I:0.0/9 ONS B3:4/11 BST MOV N7:24 N7:23 NXB GRT N7:23 1 DIV N7:23 2 N7:20 NXB LES N7:23 2 MOV N7:23 N7:20 NXB ADD N7:20 N7:32 N7:31 NXB MOV 0 N7:24 NXB ONS B3:5/15 OTE B3:6/1 BND EOR
%   I:0.0/9  LSR_TOP  "Top Part Trigger Sensor" %
%   B3:4/11  "one shot" %
%   N7:24  "check part width temporty counting" %
%   N7:23  "part width as measured at top optic part present sensor" %
%   N7:20  "1/2 top optic part width" %
%   N7:32  OPTIC_POSITION  "top optic location" %
%   N7:31  TOP_PART_LOAD_PT %
%   B3:5/15  "one shot" %
%   B3:6/1  "top part presnet one shot trailing edge" %
% Rung: 1 %
SOR XIC B18:5/11 ONS B3:7/10 OTL B9:0/1 EOR
%   B18:5/11  "Transfer bottom pass result from end of bottom conveyor" %
%   B3:7/10  "one shot" %
%   B9:0/1  "bottom of top conveyor part transfer location" %
% Rung: 2 %
SOR XIC B9:0/[N7:32] ONS B3:0/5 BST MOV 0 N7:35 NXB OTE B3:4/5 BND EOR
%   N7:32  OPTIC_POSITION  "top optic location" %
%   B3:0/5  "Transfer oneshot" %
%   N7:35  "distance since bottom part passed signal at top optic" %
%   B3:4/5  "alignment trigger for top optic" %
% Rung: 3 %
SOR OTU B9:0/[N7:32] EOR
%   N7:32  OPTIC_POSITION  "top optic location" %

